// TIA Portal V19 export
FUNCTION "ControlAutobit1" : Void   // FC50, STL
TITLE = item control 1
{ S7_Optimized_Access := 'TRUE' }
NAME : TSTOPTNK
// ****** REVISION HISTORY :
// 
// VERSION DATE       BY  DESCRIPTION
// --------------------------------------------------------------------------
// 00.00               ORIGINAL FUNCTION BLOCK
// 
// 00.01 29/5 1999   OA
// stored: AutoNumber false
   VAR_TEMP
      TEMP0 : Real;
      TEMP1 : Real;
      TEMP2 : Bool;
   END_VAR
BEGIN

NETWORK
TITLE = Product inlet valve
      A     "MY0101";
      =     "ItemStatus".Y0101.Auto;

NETWORK
TITLE = 
// S
      A     "MY0103";
      =     "ItemStatus".Y0103.Auto;

NETWORK
TITLE = Cip / steam inlet valve
      A     "MY0104";
      =     "ItemStatus".Y0104.Auto;


NETWORK
TITLE = Cooling water to jacket valve
      A     "MY0109";
      =     "ItemStatus".Y0109.Auto;

NETWORK
TITLE = 
      A     "MY0111";
      =     "ItemStatus".Y0111.Auto;


NETWORK
TITLE = 
      A     "MY0112";
      =     "ItemStatus".Y0112.Auto;


NETWORK
TITLE = 
      A     "MY0113";
      =     "ItemStatus".Y0113.Auto;


NETWORK
TITLE = Cip return / drain valve
      A     "MY0114";
      =     "ItemStatus".Y0114.Auto;


NETWORK
TITLE = Water to balance tank valve
      A     "MY0115";
      =     "ItemStatus".Y0115.Auto;
      =     "M_WATER_SUPPLY_PUMP";

NETWORK
TITLE = 
      A     "MM0139";
      =     "ItemStatus".M0139.Auto;


NETWORK
TITLE = 
      A     "MY0116";
      =     "ItemStatus".Y0116.Auto;


NETWORK
TITLE = 
      A     "MY0108";
      =     "ItemStatus".Y0108.Auto;


NETWORK
TITLE = 
      A     "MY0117";
      =     "ItemStatus".Y0117.Auto;


NETWORK
TITLE = 
      A     "MY0118";
      =     "ItemStatus".Y0118.Auto;


NETWORK
TITLE = 
      A     "MY0237";
      =     "ItemStatus".Y0237.Auto;


NETWORK
TITLE = 
      A     "MY0238";
      =     "ItemStatus".Y0238.Auto;


NETWORK
TITLE = Flush chain wash
      A     "MY0119";
      =     "ItemStatus".Y0119.Auto;


NETWORK
TITLE = 
      A     "MY0124";
      =     "ItemStatus".Y0124.Auto;

NETWORK
TITLE = 
      A     "MY0135";
      =     "ItemStatus".Y0135_NOT_USED.Auto;

NETWORK
TITLE = 
      A     "MY0136";
      =     "ItemStatus".Y0136_NOT_USED.Auto;

NETWORK
TITLE = 
      A     "MY0137";
      =     "ItemStatus".Y0137_NOT_USED.Auto;

NETWORK
TITLE = 
      A     "MY0143";
      =     "ItemStatus".Y0143.Auto;


NETWORK
TITLE = 
      A     "MY0144";
      A     "AFI";
      =     "ItemStatus".Y0144_NOT_USED.Auto;


NETWORK
TITLE = 
      A     "MY0147";
      =     "ItemStatus".Y0147.Auto;


NETWORK
TITLE = Steam valve to sterilzing
      A     "MY0148";
      =     "ItemStatus".Y0148.Auto;

NETWORK
TITLE = 
      L     "PID_TT0172/IP0157".TT0172SpDBD;
      L     15.0;
      +R;
      T     #TEMP0;
      NOP   0;

NETWORK
TITLE = Q 8.1; Output modul 1 Channel 1
      A(;
      L     "MeasuredValues".TT0172REAL;
      L     #TEMP0;
      >=R;
      );
      R     "Tag_77";
      A(;
      L     "MeasuredValues".TT0172REAL;
      L     "PID_TT0172/IP0157".TT0172SpDBD;
      <=R;
      );
      S     "Tag_77";
      NOP   0;

NETWORK
TITLE = Steam valve to injector
// Inhibit if >10degC over SP
      A     "MY0158";
      A     "Tag_77";
      =     "ItemStatus".Y0158.Auto;


NETWORK
TITLE = 
      A     "MY0545";
      =     "ItemStatus".Y0545.Auto;


NETWORK
TITLE = Relay signal to packing product availa.
      A     "M_PACK1";
      =     "ItemStatus".PACK1.Auto;


NETWORK
TITLE = 
      A     "M_PACK2";
      =     "ItemStatus".PACK2.Auto;


NETWORK
TITLE = 
      A     "M_ProdLineBeingCleaned";
      =     "ItemStatus".PACK3.Auto;

NETWORK
TITLE = Relay signal to packing product availa.
      A     "M_Time Stop CIP";
      =     "ItemStatus".PACK4.Auto;


NETWORK
TITLE = CIP Release
// CIP Release interface signal to Combi 512
      A     "M_CIP Release";
      =     "ItemStatus".AlarmLamp.Auto;
END_FUNCTION
